// TIA Portal V21 export
// export: Created 2000-01-01T00:00:00.0000000Z, ExportSetting None
FUNCTION "MCPVerify_FC_SCL_E2E" : Void   // FC903, SCL
{ S7_Optimized_Access := 'TRUE' }
// MCP 交付包：SCL 语法探针（IF/CASE/FOR/WHILE/REPEAT/转换等）
// stored: AutoNumber false, SetENOAutomatically false
   VAR_INPUT
      Enable : Bool;
      Mode : Int;
      InInt : Int;
      InReal : Real;
   END_VAR
   VAR_OUTPUT
      OutBool : Bool;
      OutInt : Int;
      OutDInt : DInt;
      OutReal : Real;
      OutWord : Word;
   END_VAR
   VAR_TEMP
      i : Int;
      acc : Int;
   END_VAR
BEGIN
   #OutBool := #Enable AND (#InInt >= 0) OR (#Mode = 2);
   #OutInt := #InInt + 1;
   #OutDInt := 0;
   #OutReal := #InReal;
   #OutWord := 16#0000;
   IF NOT #Enable THEN
     #OutInt := 0;
   ELSIF #Mode = 1 THEN
     #OutInt := #OutInt + 10;
   ELSE
     #OutInt := #OutInt + 20;
   END_IF;
   CASE #Mode OF
     0: #OutInt := 0;
     1, 2: #OutInt := #OutInt + 1;
     3..5: #OutInt := #OutInt + 3;
   ELSE
     #OutInt := -1;
   END_CASE;
   #acc := 0;
   FOR #i := 0 TO 9 DO
     #acc := #acc + #i;
   END_FOR;
   #i := 0;
   WHILE #i < 3 DO
     #acc := #acc + #i;
     #i := #i + 1;
   END_WHILE;
   REPEAT
     #acc := #acc - 1;
   UNTIL #acc <= 0
   END_REPEAT;
END_FUNCTION
